(* IEC 61131-3 sources: Industry-PLC-LLM/data/PLCBEAD_repo/PLCBEAD_PLCEmbed-main/PLC-BEAD/Source/GEB/building_TANK_VOL2, 1 file *)

(* ---- TANK_VOL2.ST ---- *)
FUNCTION TANK_VOL2:REAL

	VAR_INPUT
		TR :	REAL;
		H :	REAL;
	END_VAR

	TANK_VOL2 := 3.14159265358979323846264338327950288 * H * H * (TR - H / 3.0);

END_FUNCTION

PROGRAM program0
  VAR
    TR :	REAL;
	H :	REAL;
    CEIL5_OUT : REAL;
  END_VAR

  CEIL5_OUT := TANK_VOL2(TR, H);
END_PROGRAM
